// TIA Portal V20 export
TYPE "LER_typeMobileRFIDCommands"
// stored: Access Published
   STRUCT
      ResetReq : Bool;
      resultRFIDReset : Bool;
   END_STRUCT;
END_TYPE
